// TIA Portal V19 export
ORGANIZATION_BLOCK "Diagnostic error interrupt"   // OB82, STL, DiagnosticErrorInterrupt
{ S7_Optimized_Access := 'FALSE' }
   VAR_TEMP
      EV_CLASS : Byte;   // 16#39: Event class 3, Entering event state, Internal fault event
      FLT_ID : Byte;   // Fault identifier
      PRIORITY : Byte;   // Priority of OB Execution
      OB_NUMBR : Byte;   // OB number
      RESERVED_1 : Byte;   // Reserved for system
      IO_FLAG : Byte;   // 16#54:input, 16#55:output, 16#0:not available
      MDL_ADDR : Word;   // Hardware identifier
      MDL_DEFECT : Bool;   // Module defective
      INT_FAULT : Bool;   // Internal fault
      EXT_FAULT : Bool;   // External fault
      PNT_INFO : Bool;   // Channel fault
      EXT_VOLTAGE : Bool;   // External voltage low
      FLD_CONNCTR : Bool;   // Field wiring connector missing
      NO_CONFIG : Bool;   // Module has no configuration data
      CONFIG_ERR : Bool;   // Module has configuration error
      MDL_TYPE : Byte;   // Type of module
      SUB_MDL_ERR : Bool;   // Sub-Module is missing or has error
      COMM_FAULT : Bool;   // Communication fault
      MDL_STOP : Bool;   // Module is stopped
      WTCH_DOG_FLT : Bool;   // Watch dog timer stopped module
      INT_PS_FLT : Bool;   // Internal power supply fault
      PRIM_BATT_FLT : Bool;   // Primary battery is in fault
      BCKUP_BATT_FLT : Bool;   // Backup battery is in fault
      RESERVED_2 : Bool;   // Reserved for system
      RACK_FLT : Bool;   // Rack fault, only for bus interface module
      PROC_FLT : Bool;   // Processor fault
      EPROM_FLT : Bool;   // EPROM fault
      RAM_FLT : Bool;   // RAM fault
      ADU_FLT : Bool;   // ADU fault
      FUSE_FLT : Bool;   // Fuse fault
      HW_INTR_FLT : Bool;   // Hardware interrupt input in fault
      RESERVED_3 : Bool;   // Reserved for system
      DATE_TIME : Date_And_Time;   // Date and time OB82 started
   END_VAR
BEGIN
END_ORGANIZATION_BLOCK
